# EPICS substitutions: elioApp/Db/EL2808.substitutions
file EL2808.template { pattern
{ CHAN	}
{ 1	}
{ 2	}
{ 3	}
{ 4	}
{ 5	}
{ 6	}
{ 7	}
{ 8	}
}
